# EPICS StreamDevice protocol: laudaRE2xxApp/protocol/lRE2xx.proto
##################################################
#
# Protocol File
#
# Protocol file for Lauda Ecoline Staredition RE2xx
# Diamond Light Source, Oct 2008
#
# NOTES:
#
#
#
##################################################

##################################################
# General Settings
##################################################

Terminator = "\r\n";
ReplyTimeout = 1000;

###################################################
# Get functions
###################################################

# /// Read water bath temperature
getTemp {
   ExtraInput = Ignore;
   out "IN_PV_00";
   in "%f";
}

# /// Read over temperature status
getStatus {
   ExtraInput = Ignore;
   seperator = "";
   out "STAT";
   in "%1d";
}

###################################################
# Set functions
###################################################

# /// Set the setpoint for water temperature (temperature must be specific format (up to 3 digits before decimal point and up to 2 digits after decimal point).
setTemp {
   out "OUT_SP_00_%f";
}

#############################################################
# Generic protocol
############################################################

# /// Use this send any command and get back the response (max 39 chars).
gen {
    ExtraInput = Ignore;
    out "%s";
    in "%39c"
}
